(* IEC 61131-3 sources: programs/VI-54/VI-54_20171205/VI-54_20171205/Stations/Screen/LseClass170718/Class/DiagnoseHelpClass, 1 file *)

(* ---- DiagnoseHelpClass.st ---- *)
(*!
<Class
	Name               = "DiagnoseHelpClass"
	Revision           = "1.0"
	RealtimeTask       = "false"
	CyclicTask         = "false"
	BackgroundTask     = "false"
	Sigmatek           = "false"
	OSInterface        = "false"
	HighPriority       = "false"
	Automatic          = "false"
	UpdateMode         = "Prescan"
	SharedCommandTable = "true"
	Objectsize         = "(540,360)"
	Comment            = "helping class for working with the PLC">
	<Channels>
		<Server Name="ClassSvr" Visualized="false" Initialize="false" WriteProtected="true" Retentive="false" Comment="class server"/>
		<Server Name="OpenDiagnose" Visualized="true" Initialize="false" WriteProtected="false" Retentive="false" Comment="write() will open the diagnosis"/>
		<Server Name="Reboot" Visualized="true" Initialize="false" WriteProtected="false" Retentive="false" Comment="write() will cause a plc REBOOT"/>
		<Server Name="Reset" Visualized="true" Initialize="false" WriteProtected="false" Retentive="false" Comment="write() will cause a plc RESET"/>
		<Server Name="ResetRun" Visualized="true" Initialize="false" WriteProtected="false" Retentive="false" Comment="write() will cause ResetRunApp"/>
		<Client Name="toOsKernel" Required="false" Internal="false" Comment="object channel to toOsKernel (don&apos;t connect)"/>
	</Channels>
	<RevDoku>
		<Owner Company="Sigmatek"/>
		<Dokumentation Revision="1.0" Date="2015-09-22" Company="Sigmatek" Description="Creation."/>
	</RevDoku>
</Class>
*)
DiagnoseHelpClass : CLASS
  //Servers:
	ClassSvr 	: SvrChCmd_DINT;
	Reset 	: SvrCh_DINT;
	Reboot 	: SvrCh_DINT;
	ResetRun 	: SvrCh_DINT;
	OpenDiagnose 	: SvrCh_DINT;
  //Clients:
	toOsKernel 	: CltChCmd__OSKernel;
  //Variables:
  //Functions:

	FUNCTION VIRTUAL GLOBAL Reset::Write
		VAR_INPUT
			input (EAX) 	: DINT;
		END_VAR
		VAR_OUTPUT
			result (EAX) 	: DINT;
		END_VAR;

	FUNCTION VIRTUAL GLOBAL Reboot::Write
		VAR_INPUT
			input (EAX) 	: DINT;
		END_VAR
		VAR_OUTPUT
			result (EAX) 	: DINT;
		END_VAR;

	FUNCTION VIRTUAL GLOBAL ResetRun::Write
		VAR_INPUT
			input (EAX) 	: DINT;
		END_VAR
		VAR_OUTPUT
			result (EAX) 	: DINT;
		END_VAR;

	FUNCTION VIRTUAL GLOBAL OpenDiagnose::Write
		VAR_INPUT
			input (EAX) 	: DINT;
		END_VAR
		VAR_OUTPUT
			result (EAX) 	: DINT;
		END_VAR;
  //Tables:
	FUNCTION @STD
		VAR_OUTPUT
			ret_code	: CONFSTATES;
		END_VAR;
	FUNCTION GLOBAL TAB @CT_;
END_CLASS;

#pragma usingLtd _OSKernel

FUNCTION VIRTUAL GLOBAL DiagnoseHelpClass::Reset::Write
	VAR_INPUT
		input (EAX) 	: DINT;
	END_VAR
	VAR_OUTPUT
		result (EAX) 	: DINT;
	END_VAR

	Reset := input;

  toOsKernel.Reset();

	result := Reset;

END_FUNCTION

FUNCTION VIRTUAL GLOBAL DiagnoseHelpClass::Reboot::Write
	VAR_INPUT
		input (EAX) 	: DINT;
	END_VAR
	VAR_OUTPUT
		result (EAX) 	: DINT;
	END_VAR

	Reboot := input;

  toOsKernel.Reboot();

	result := Reboot;

END_FUNCTION

FUNCTION VIRTUAL GLOBAL DiagnoseHelpClass::ResetRun::Write
	VAR_INPUT
		input (EAX) 	: DINT;
	END_VAR
	VAR_OUTPUT
		result (EAX) 	: DINT;
	END_VAR

	ResetRun := input;
  toOsKernel.ResetRunApp();
	result := ResetRun;

END_FUNCTION

FUNCTION VIRTUAL GLOBAL DiagnoseHelpClass::OpenDiagnose::Write
	VAR_INPUT
		input (EAX) 	: DINT;
	END_VAR
	VAR_OUTPUT
		result (EAX) 	: DINT;
	END_VAR

	OpenDiagnose := input;
  InsertCmd(CMD_DIAGNOSTIC, 0, 0);
	result := OpenDiagnose;

END_FUNCTION
